PROGRAM CamTable
VAR
	bLoadPoints: BOOL;
	bCamInit			: BOOL;

	arCamTable			: ARRAY [0..iNumPts, 0..1] OF LREAL;
	CamTblSelect		: MC_CamTableSelect;
	CamTableRef			: MC_Cam_Ref;
	ST_CamInOptions_V2	: ST_CamInOptions_V2;

	CamIn_v2			: MC_CamIn_V2;
	CamOut				: MC_CamOut;
	bCamIn				: BOOL;

	osrTblSlct			: F_TRIG;
	bPeriodic			: BOOL;

	iInterpType			: UINT :=1;		// start with spline

	iSelX				: INT;			// selected visualization col
	iSelY				: INT;			// selected visualization row 
	
END_VAR

VAR CONSTANT
	iNumPts 			: UDINT := 5;
END_VAR

Cam_Setup();

IF bLoadPoints THEN
	LoadPoints();
	bLoadPoints:=FALSE;
END_IF

IF bCamInit THEN
	Cam_Init();
	bCamInit := FALSE;
END_IF

ACTION Cam_Init:

CamTableRef.pArray := ADR(arCamTable);
CamTableRef.ArraySize := SIZEOF(arCamTable);

CamTableRef.TableType := MC_TABLETYPE_EQUIDISTANT ;

CamTableRef.NoOfRows := iNumPts;
CamTableRef.NoOfColumns := 2;
ST_CamInOptions_V2.CamOperationMode:=CAMOPERATIONMODE_ADDITIVE;


CASE iInterpType OF
0:
	ST_CamInOptions_V2.InterpolationType:=MC_INTERPOLATIONTYPE_LINEAR;
1:
	ST_CamInOptions_V2.InterpolationType:=MC_INTERPOLATIONTYPE_SPLINE;
2:
	ST_CamInOptions_V2.InterpolationType:=MC_INTERPOLATIONTYPE_SLIDINGSPLINE;
END_CASE
END_ACTION

ACTION Cam_Setup:
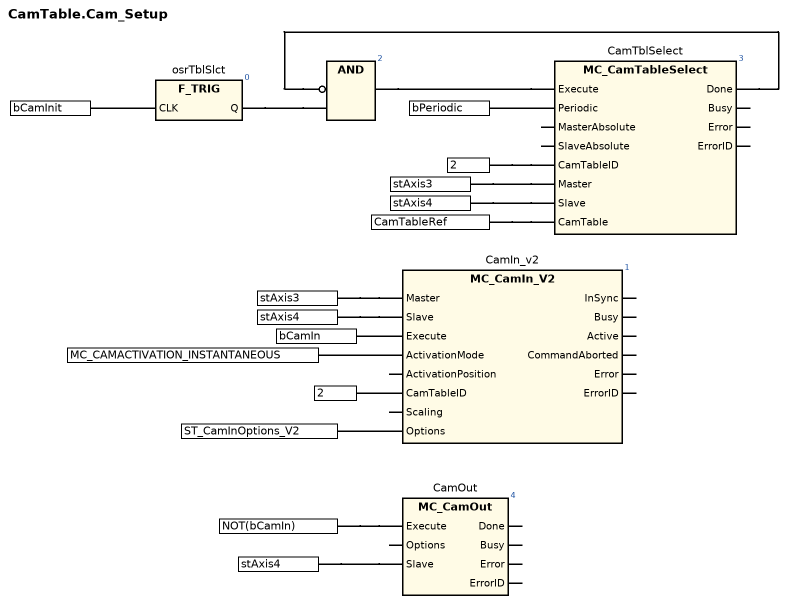
osrTblSlct(CLK := bCamInit); // F_TRIG
CamIn_v2(
    Master := stAxis3,
    Slave := stAxis4,
    Execute := bCamIn,
    ActivationMode := MC_CAMACTIVATION_INSTANTANEOUS,
    CamTableID := 2,
    Options := ST_CamInOptions_V2); // MC_CamIn_V2
CamTblSelect(
    Execute := NOT CamTblSelect.Done AND osrTblSlct.Q,
    Periodic := bPeriodic,
    CamTableID := 2,
    Master := stAxis3,
    Slave := stAxis4,
    CamTable := CamTableRef); // MC_CamTableSelect
CamOut(Execute := NOT(bCamIn), Slave := stAxis4); // MC_CamOut
END_ACTION

ACTION LoadPoints:
arCamTable[0,0] := 0;
arCamTable[0,1] := 0;

arCamTable[1,0] := 250;
arCamTable[1,1] := 500;

arCamTable[2,0] := 500;
arCamTable[2,1] := 1000;

arCamTable[3,0] := 750;
arCamTable[3,1] := 500;

arCamTable[4,0] := 1000;
arCamTable[4,1] := 0;
END_ACTION

END_PROGRAM

(* stored: Version 1.1.0.1, ProductVersion 3.1.4024.11
   POU CamTable: Id {68bfe7fc-b7e0-4b43-959b-c77649601557}, SpecialFunc None
   Action Cam_Init: Id {c90bac94-e1cc-496b-a046-820cbbf8b35d}
   Action Cam_Setup: Id {153c0b49-a37f-466c-b87f-9cb02c6310e6}
   Action LoadPoints: Id {50960435-1b5d-4fa1-9681-48751e9d3272} *)
